FUNCTION_BLOCK FB_Sum
VAR_INPUT
	one : UINT;
	two : UINT;
END_VAR
VAR_OUTPUT
	result : UINT;
END_VAR

result := one + two;

END_FUNCTION_BLOCK

(* stored: Version 1.1.0.1, ProductVersion 3.1.4022.18
   POU FB_Sum: Id {8328f7d8-1dbc-4e08-98b0-eb6438d2b355}, SpecialFunc None *)
